// SIMATIC S7-200 project (STEP 7-Micro/WIN), CPU 224XP REL 02.01

SYMBOL_TABLE USUARIO1
INTERRUPTOR      I0.0
LAMPARA_PARO     Q0.0
LAMPARA_M1       Q0.1
LAMPARA_M2       Q0.2
END_SYMBOL_TABLE

ORGANIZATION_BLOCK PRINCIPAL:OB1
TITLE=COMENTARIOS DEL PROGRAMA
BEGIN
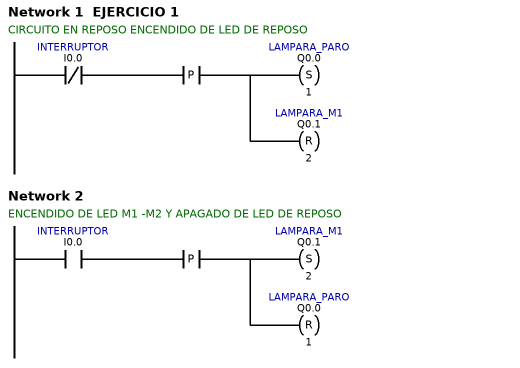
Network 1 // EJERCICIO 1
// CIRCUITO EN REPOSO ENCENDIDO DE LED DE REPOSO
// (network saved uncompiled; LAD cells follow)
// row 0: c0 -|/|- INTERRUPTOR:I0.0  c1 -|P|-  v  c2 -(S) LAMPARA_PARO:Q0.0, 1
// row 1: c1 ^  c2 -(R) LAMPARA_M1:Q0.1, 2
Network 2
// ENCENDIDO DE LED M1 -M2 Y APAGADO DE LED DE REPOSO
// (network saved uncompiled; LAD cells follow)
// row 0: c0 -| |- INTERRUPTOR:I0.0  c1 -|P|-  v  c2 -(S) LAMPARA_M1:Q0.1, 2
// row 1: c1 ^  c2 -(R) LAMPARA_PARO:Q0.0, 1
END_ORGANIZATION_BLOCK
